(* PLC project 117_1_V0.5.project, CODESYS CODESYS V3.5 SP17 Patch 3 *)
(* stored: creationDateTime 1970-01-01T00:00:00, modificationDateTime 2026-03-26T18:14:32.4070562 *)

PROGRAM MAIN
  VAR
    TimeManagerEx : TimeManager;  (* Блок с данными о времени *)
    InputManagerEx : InputManager;  (* Блок с данными входных сигналов *)
    StandLogicEx : StandLogic;  (* Логика управления стэндом *)
    ServoDriverEx : SM3ServoDriver;  (* Блок туправления сервоприводом *)
    PIDControllerEx : BasicPIDController;  (* Блок пегулятора *)
    OutputManagerEx : OutputManager;  (* Блок с данными выходных сигналов *)
  END_VAR

            // Данные задачи
TimeManagerEx();

// Входные данные
InputManagerEx();

// Логика управления стэндом
StandLogicEx(
		TimeManager			:= TimeManagerEx,
		InputManager		:= InputManagerEx,
		PIDController		:= PIDControllerEx,
		ServoDriver			:= ServoDriverEx,
 		OutputManager		:= OutputManagerEx);	
			
// Регулятор		
PIDControllerEx();
	
// Сервопривод	
ServoDriverEx(TimeManager := TimeManagerEx);		
		
// Пишем выходные данные		
OutputManagerEx();



          
END_PROGRAM
